# EPICS alarm handler configuration: alh_files/mgnt_dmp1_bend.alhConfig
GROUP NULL BEND:DMP1:MG01
   $COMMAND edm -x -eolc -noedit mgnt_dmp1_bend.edl
$ALIAS BEND
$GUIDANCE
DMP1 BEND
   Group Name: BEND:DMP1:MG01
   Summary PV:  BEND:DMP1:MG01:STATSUMY
$END

GROUP BEND:DMP1:MG01  BEND:DMP1:400
   $COMMAND edm -x -eolc -noedit -m "DEV=BEND:DMP1:400" mgnt_unit.edl
CHANNEL    BEND:DMP1:400    BEND:DMP1:400:STATMSG   -----
   $FORCEPV BEND:DMP1:400:STATMSGSV -DATL 1 0
